TYPE FB_TcpClient_State :
(
	UNDEFINIERT := 0,
	GETRENNT,
	VERBINDEN,
	VERBUNDEN,
	SENDEN,
	MESSAGE_AUSLESEN,
	TRENNEN,	
	
	
	ERROR_HANDLER
);
END_TYPE

(* stored: Version 1.1.0.1, ProductVersion 3.1.4018.5
   DUT FB_TcpClient_State: Id {4727be23-725f-4636-aecf-0f7cc85fefdb} *)
